{attribute 'GeneratedUsingTerminal: EL9576-0000-0019'}
{attribute addProperty BoxType "EL9576-0000-0019"}
{attribute addProperty Id "EtcSlaveTerminalBaseBCT_InputsAT %I*BCT_Inputs_4B98789517WcStateAT %I*WcState_9091E0EB2InfoDataAT %I*InfoData_32EB74EA10"}
{attribute addProperty CRC "2273633773"}
{attribute addProperty Size "29"}
TYPE EL9576_8784E5ED EXTENDS EtcSlaveTerminalBase :
STRUCT
	{attribute addProperty Name "BCT_Inputs"}
	BCT_Inputs : BCT_Inputs_4B987895;
	{attribute addProperty Name "WcState"}
	WcState : WcState_9091E0EB;
	{attribute addProperty Name "InfoData"}
	InfoData : InfoData_32EB74EA;
END_STRUCT
END_TYPE

(* stored: Version 1.2.0.0, ProductVersion 3.1.4024.9
   DUT EL9576_8784E5ED: Id {e7d987b3-61ea-49c9-b529-f3e377c88fea} *)
